// TIA Portal V16 export
// export: Created 2022-11-14T17:35:45.4169233Z, ExportSetting WithDefaults, DisplayName Totally Integrated Automation Portal, DisplayVersion V16, DisplayName TIA Portal Version Control Interface, DisplayVersion V16, DisplayName TIA Portal Openness, DisplayVersion V16, DisplayName STEP 7 Professional, DisplayVersion V16, DisplayName STEP 7 Safety, DisplayVersion V16, DisplayName WinCC Advanced, DisplayVersion V16
DATA_BLOCK "U201_Process_Data"   // DB211
VERSION : 0.1
// stored: AutoNumber false, InstanceOfName Inverter_Process_Data, InstanceOfType FB
"Inverter_Process_Data"
   // VAR_INPUT
   //    control_word : Word;
   //    setpoint : Real;
   //    RD_address : HW_SUBMODULE;
   //    WR_address : HW_SUBMODULE;
   //    ref_quantity : Struct
   //       speed_p2000 : Real;
   //       current_p2002 : Real;
   //       torque_p2003 : Real;
   //    END_STRUCT;
   // END_VAR
   // VAR_OUTPUT
   //    status_word : Word;
   //    actual_speed : Real;
   //    actual_current : Real;
   //    actual_torque : Real;
   //    actual_alarm : Word;
   //    actual_fault : Word;
   //    RETVAL_RD : Word;
   //    RETVAL_WR : Word;
   // END_VAR
BEGIN
END_DATA_BLOCK
